//设备报警处理
FUNCTION error_Trigger : BOOL
VAR_INPUT
	errorID					:DINT;//error id
END_VAR
VAR
END_VAR

IF g_Max_Data_Elements<=gError_hTable.nCount THEN//哈希表内容超过100条，直接返回
	RETURN;
END_IF
gError_fbTable.A_Lookup(key:=TO_DWORD(errorID),hTable:=gError_hTable);//从哈希表中查询是否有正在报警的id
IF gError_fbTable.bOk THEN//如果有，直接返回，不再报警该id；如果无，则添加到哈希表中，并报警提示
	//value:= gError_fbTable.getValue;
	RETURN;//已经报警过该错误
ELSE
	(* Entry not found *)
	gError_fbTable.A_Add(key:=TO_DWORD(errorID),putValue :=TO_UDINT(errorID), hTable:=gError_hTable);
END_IF
//print之前，先进行ErrorMonitor将错误内容进行分配；如果错误内容写死，可以不用这么写
errorMonitor();
error_Printf(errorID);

IF g_d_ErrorBegin<=errorID AND errorID<=g_d_ErrorEnd THEN
	CASE gErrorARRAY[errorID].eErrLevel OF
		Error_Level_0:
			//gErrorARRAY[errorID].bError:=TRUE;
			IF gAutoRunningFlag THEN
				//PLC_MainSW.appendSend(0,0,E_CmdID_SW.SW_Error,0.0,0.0,0.0,0.0,gErrorARRAY[errorID].eErrLevel,gErrorARRAY[errorID].uErrID,gErrorARRAY[errorID].sErrTXT);
				//PLC_MainSW.appendSend(0,0,E_CmdID_SW.SW_Error,0.0,0.0,0.0,0.0,0.0,ErrCodeProcess(errorID),'');
				//PLC_MainSW.appendSend(TO_STRING(ErrCodeProcess(errorID)));
			END_IF
		Error_Level_1:
			//gErrorARRAY[errorID].bError:=TRUE;
			IF gAutoRunningFlag THEN
				//PLC_MainSW.appendSend(0,0,E_CmdID_SW.SW_Error,0.0,0.0,0.0,0.0,gErrorARRAY[errorID].eErrLevel,gErrorARRAY[errorID].uErrID,gErrorARRAY[errorID].sErrTXT);
				//PLC_MainSW.appendSend(TO_STRING(ErrCodeProcess(errorID)));
			END_IF
		Error_Level_2:
			//gErrorARRAY[errorID].bError:=TRUE;
			IF gAutoRunningFlag THEN
				//PLC_MainSW.appendSend(0,0,E_CmdID_SW.SW_Error,0.0,0.0,0.0,0.0,gErrorARRAY[errorID].eErrLevel,gErrorARRAY[errorID].uErrID,gErrorARRAY[errorID].sErrTXT);
				//PLC_MainSW.appendSend(TO_STRING(ErrCodeProcess(errorID)));
			END_IF
		Error_Level_3:
			gErrorARRAY[errorID].bError:=TRUE;
			IF gAutoRunningFlag THEN
				//PLC_MainSW.appendSend(0,0,E_CmdID_SW.SW_Error,0.0,0.0,0.0,0.0,gErrorARRAY[errorID].eErrLevel,gErrorARRAY[errorID].uErrID,gErrorARRAY[errorID].sErrTXT);
				//PLC_MainSW.appendSend(TO_STRING(ErrCodeProcess(errorID)));
			END_IF
		Error_Level_4:
			gErrorARRAY[errorID].bError:=TRUE;
			IF gAutoRunningFlag THEN
				//PLC_MainSW.appendSend(0,0,E_CmdID_SW.SW_Error,0.0,0.0,0.0,0.0,gErrorARRAY[errorID].eErrLevel,gErrorARRAY[errorID].uErrID,gErrorARRAY[errorID].sErrTXT);
				//PLC_MainSW.appendSend(TO_STRING(ErrCodeProcess(errorID)));
			END_IF
	END_CASE
END_IF

END_FUNCTION

(* stored: Version 1.1.0.1, ProductVersion 3.1.4024.4
   POU error_Trigger: Id {bc2485ac-ad7a-4601-9a6f-f9dccf8c5295}, SpecialFunc None *)
